TYPE TimeChannelParameters :
STRUCT
	TC01: TimeChannel1CH_Data := ( Day := TimerDays.Monday, OffTime := 2400 );
	TC02: TimeChannel1CH_Data := ( Day := TimerDays.Tuesday, OffTime := 2400 );
	TC03: TimeChannel1CH_Data := ( Day := TimerDays.Wednesday, OffTime := 2400 );
	TC04: TimeChannel1CH_Data := ( Day := TimerDays.Thursday, OffTime := 2400 );
	TC05: TimeChannel1CH_Data := ( Day := TimerDays.Friday, OffTime := 2400 );
	TC06: TimeChannel1CH_Data := ( Day := TimerDays.Saturday, OffTime := 2400 );
	TC07: TimeChannel1CH_Data := ( Day := TimerDays.Sunday, OffTime := 2400 );
	TC11: TimeChannel1CH_Data := ( Day := TimerDays.Monday );
	TC12: TimeChannel1CH_Data := ( Day := TimerDays.Tuesday );
	TC13: TimeChannel1CH_Data := ( Day := TimerDays.Wednesday );
	TC14: TimeChannel1CH_Data := ( Day := TimerDays.Thursday );
	TC15: TimeChannel1CH_Data := ( Day := TimerDays.Friday );
	TC16: TimeChannel1CH_Data := ( Day := TimerDays.Saturday );
	TC17: TimeChannel1CH_Data := ( Day := TimerDays.Sunday );
	TC21: TimeChannel1CH_Data := ( Day := TimerDays.Monday, Speed := 2 );
	TC22: TimeChannel1CH_Data := ( Day := TimerDays.Tuesday, Speed := 2 );
	TC23: TimeChannel1CH_Data := ( Day := TimerDays.Wednesday, Speed := 2 );
	TC24: TimeChannel1CH_Data := ( Day := TimerDays.Thursday, Speed := 2 );
	TC25: TimeChannel1CH_Data := ( Day := TimerDays.Friday, Speed := 2 );
	TC26: TimeChannel1CH_Data := ( Day := TimerDays.Saturday, Speed := 2 );
	TC27: TimeChannel1CH_Data := ( Day := TimerDays.Sunday, Speed := 2 );
	Q: BOOL; // Result of the time channels
	HighSpeed: BOOL; // Speed result of the time channels
END_STRUCT
END_TYPE

(* stored: Version 1.1.0.1, ProductVersion 3.1.4024.6
   DUT TimeChannelParameters: Id {510b2f36-2e49-4977-925d-903649d03032} *)
